// LS Electric XG5000 project: project
// PLC LSPLC
// module base 0 slot 0: 입출력 모듈:XBC-DN/DP32H (DC 24V 입력, 트랜지스터 출력 32점 (싱크출력/소스출력))

PROGRAM NewProgram (task: 스캔 프로그램)

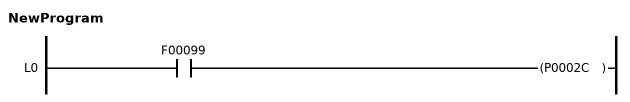
; L0
LOAD      F00099
OUT       P0002C